# EPICS autosave request: rsfsxApp/Db/rsfsv_settings.req
# This file specifies which PVs of the corresponding database should be saved.
file "rsfsx_settings.req",                P=$(P),  R=$(R)

$(P)$(R)FiltType-Sel
$(P)$(R)AutoFreq-Cmd
$(P)$(R)AutoLvl-Cmd
$(P)$(R)AutoAll-Cmd
$(P)$(R)SaveTrig
